TYPE E_MainStateMachine :
(
	eMainSM_BasicInit 						:= 0,
	eMainSM_TempInit,
	eMainSM_MParamLoad,
	eMainSM_PParamLoad,
	eMainSM_SupParamLoad,
	eMainSM_StartUp,
	eMainSM_Idle
);
END_TYPE

(* stored: Version 1.1.0.1, ProductVersion 3.1.4024.12
   DUT E_MainStateMachine: Id {307774db-ccd3-4d90-aa67-0b9aed463f8b} *)
